FUNCTION_BLOCK DigitalController
  (* Standard: 61499-2 *)
  (* Version 0.1, 2015-00-11, syy, syy-PC *)
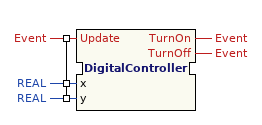
  EVENT_INPUT
    Update WITH x, y;
  END_EVENT
  EVENT_OUTPUT
    TurnOn;
    TurnOff;
  END_EVENT
  VAR_INPUT
    x : REAL;
    y : REAL;
  END_VAR
  VAR
    control : REAL;
    timer : REAL;
  END_VAR
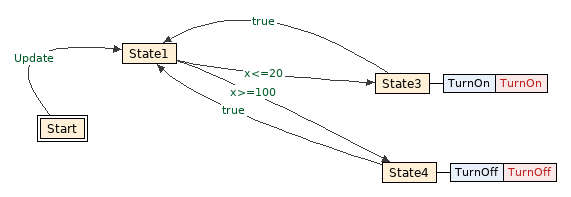
  EC_STATES
    Start;
    State1;
    State3 : TurnOn -> TurnOn;
    State4 : TurnOff -> TurnOff;
  END_STATES
  EC_TRANSITIONS
    Start TO State1 := Update;
    State1 TO State3 := x<=20;
    State1 TO State4 := x>=100;
    State3 TO State1 := true;
    State4 TO State1 := true;
  END_TRANSITIONS
  ALGORITHM RandomChoice IN C:
me->timer=0;

/* Intializes random number generator */
srand(time(NULL));

me->control = rand() % 2 ;
//printf("control : %d\n", me->control);
  END_ALGORITHM
  ALGORITHM Wait IN C:
//printf("signal sent\n");
wait(10);
//me->timer++;
  END_ALGORITHM
  ALGORITHM TurnOn IN C:
printf("Signal sent : turn on the burner |  Temperature : %f\n", me->x);
wait(10);
  END_ALGORITHM
  ALGORITHM TurnOff IN C:
printf("Signal sent : turn off the burner |  Temperature : %f\n", me->x);
wait(10);
  END_ALGORITHM
  ALGORITHM printing IN C:
printf("x=%f\n", me->x);
  END_ALGORITHM
END_FUNCTION_BLOCK
